// TwinCAT 3 PLC project SideEffectPLC
// ProgramVersion: 3.1.4026.20
// CompilerDefines: VISU_USEPROPERTYINFO
// libraries:
//   Tc2_Standard, * (Beckhoff Automation GmbH)
//   Tc2_System, * (Beckhoff Automation GmbH)
//   Tc2_Utilities, * (Beckhoff Automation GmbH)
//   VisuSymbols, 4.5.0.0 (System)
// project tree:
//   DUTs/ DUT_Climate_Monoid.TcDUT, DUT_Effect.TcDUT (not stored), DUT_Effect_Monoid.TcDUT, DUT_Effect_Monoid_1.TcDUT, DUT_Humidity_Monoid.TcDUT, DUT_Pressure_Monoid.TcDUT (not stored), ENUM_Effect_Type.TcDUT (not stored)
//   / GlobalTextList.TcGTLO, PlcTask.TcTTO, Visualization Manager.TcVMO (not stored)
//   GVLs/ GVL.TcGVL (not stored)
//   POUs/Constructors/ FC_AlarmEffect.TcPOU (not stored), FC_IoTEffect.TcPOU (not stored), FC_LogEffect.TcPOU (not stored), FC_ValveEffect.TcPOU (not stored), FC_StopInputEffect.TcPOU (not stored), FC_StartInputEffect.TcPOU (not stored), FC_ResetInputEffect.TcPOU (not stored), FC_TickInputEffect.TcPOU (not stored)
//   POUs/ Control_LOOP.TcPOU (not stored), SideEffect_LOOP.TcPOU (not stored), Simulation_LOOP.TcPOU (not stored)
//   POUs/Monoid/ FC_CombineClimate.TcPOU (not stored), FC_CombineHumidity.TcPOU (not stored), FC_CombinePressure.TcPOU (not stored), FC_EmptyHumidity.TcPOU (not stored), FC_EmptyPressure.TcPOU (not stored), FC_CombineEffects.TcPOU (not stored), FC_EmptyEffect.TcPOU (not stored)
//   POUs/PLCLogic/ FB_HumidityLogic.TcPOU (not stored), FB_PressureLogic.TcPOU (not stored), FB_SimpleLogic.TcPOU (not stored)
//   POUs/Simulation/ FB_PlantSimulator.TcPOU (not stored)
//   VISUs/ Visualization.TcVIS

CONFIGURATION SideEffectPLC
    RESOURCE PLC ON TwinCAT3
        TASK PlcTask(INTERVAL := T#10ms, PRIORITY := 20);
        PROGRAM SideEffect_LOOP WITH PlcTask : SideEffect_LOOP;
        PROGRAM Simulation_LOOP WITH PlcTask : Simulation_LOOP;
        PROGRAM Control_LOOP WITH PlcTask : Control_LOOP;
    END_RESOURCE
END_CONFIGURATION

// ---- DUTs/DUT_Climate_Monoid.TcDUT
// 这是一个典型的 Product Monoid, 将多个子幺半群独立地结合在一起
// 纵向扩展：每增加一个控制域，只需添加一个新字段 + 对应的 Combine 函数
TYPE DUT_Climate_Monoid :
STRUCT
	Temp     : DUT_Effect_Monoid;       // 温度控制 (Free Monoid)
	Hum      : DUT_Humidity_Monoid;     // 湿度控制 (Sum Monoid)
	Pressure : DUT_Pressure_Monoid;     // 压力监控 (Max Monoid) — 纵向扩展新增
END_STRUCT
END_TYPE

// ---- DUTs/DUT_Effect_Monoid.TcDUT
TYPE DUT_Effect_Monoid :
STRUCT
	Count   : INT := 0;
    Effects : ARRAY[1..20] OF DUT_Effect;
END_STRUCT
END_TYPE

// ---- DUTs/DUT_Effect_Monoid_1.TcDUT
TYPE DUT_Effect_Monoid_1 :
STRUCT
	Count   : INT := 0;
    Effects : ARRAY[1..20] OF DUT_Effect;
END_STRUCT
END_TYPE

// ---- DUTs/DUT_Humidity_Monoid.TcDUT
// 模拟加法幺半群：存储累计喷洒量的单维度载体
TYPE DUT_Humidity_Monoid :
STRUCT
	SprayAmount : REAL := 0.0; // The total volume of moisture to spray
END_STRUCT
END_TYPE

// ---- GlobalTextList.TcGTLO
TEXTLIST GlobalTextList
  592 = '%s'
  184 = 'Reset'
  492 = 'Start'
  75 = 'Stop'
END_TEXTLIST

// ---- VISUs/Visualization.TcVIS
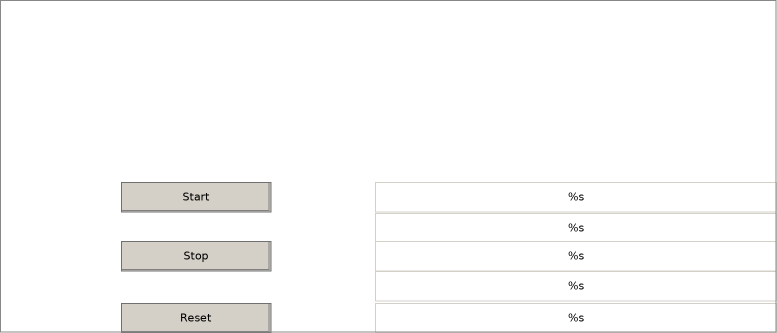
VISUALIZATION Visualization  // 777x333
    Button (121,182 150x30), "Start"
        tap GVL.Inbox_IoT_SoftStart
    Button (121,241 150x30), "Stop"
        tap GVL.Inbox_IoT_SoftStop
    Button (121,303 150x30), "Reset"
        tap GVL.Inbox_IoT_SoftReset
    Textfield (375,182 402x30), "%s", text variable: GVL.HMI_Logs[1]
    Textfield (375,213 402x30), "%s", text variable: GVL.HMI_Logs[2]
    Textfield (375,241 402x30), "%s", text variable: GVL.HMI_Logs[3]
    Textfield (375,271 402x30), "%s", text variable: GVL.HMI_Logs[4]
    Textfield (375,303 402x30), "%s", text variable: GVL.HMI_Logs[5]
END_VISUALIZATION
